TYPE ST_SafetyDoor_IO :
STRUCT
	stHwIn AT%I* : ST_SafetyDoor_IN;
	stHwOut	AT%Q* : ST_SafetyDoor_OUT;
END_STRUCT
END_TYPE

(* stored: Version 1.1.0.1
   DUT ST_SafetyDoor_IO: Id {a3da1635-c954-4c79-a888-a438f0da517b} *)
